FUNCTION_BLOCK FB_Estacion
VAR_INPUT
END_VAR
VAR_OUTPUT
	//Parametros de salida
	PaleCodigo: BYTE;
END_VAR
VAR
	//Entradas comunes
	PulsadorEmergencia AT %I*: BOOL;
    SelectorManual AT %I*: BOOL;
    PulsadorMarcha AT %I*: BOOL;
    PulsadorParada AT %I*: BOOL := TRUE; // Contacto normalmente cerrado
    EstacionConectada AT %I*: BOOL := TRUE;
    DetectorPresion AT %I*: BOOL := TRUE;
	
	PalePresencia AT %I*: BOOL;
    PaleCodigoBit0 AT %I*: BOOL;
    PaleCodigoBit1 AT %I*: BOOL;
    PaleCodigoBit2 AT %I*: BOOL;
	
	//Entradas específicas
	DescargadorDetras AT %I*: BOOL;
	DescargadorDelante AT %I*: BOOL;
	VerticalArriba AT %I*: BOOL;
	VerticalAbajo AT %I*: BOOL;
	VerificadorArriba AT %I*: BOOL;
	VerificadorAbajo AT %I*: BOOL;
	DesplazadorDetras AT %I*: BOOL;
	AlimentadorDetras AT %I*: BOOL;
	AlimentadorDelante AT %I*: BOOL;
	VacioDescargador AT %I*: BOOL;
	PresenciaBaseAlimentador AT %I*:BOOL;
	
	//Salidas comunes
	DesconectaEstacion AT %Q*: BOOL;
    LamparaAlarma AT %Q*: BOOL;
    LamparaMarcha AT %Q*: BOOL;
	LamparaFaltaMaterial AT %Q*: BOOL;
    AvisadorSonoro AT %Q*: BOOL;

    CintaMotorActiva AT %Q*: BOOL;
    CintaMotorInvierte AT %Q*: BOOL;
    CintaRetenedorBaja AT %Q*: BOOL;
    CintaSeparadorSube AT %Q*: BOOL;
	
	//Salidas específicas
	DescargadorAtras AT %Q*: BOOL;
	DescargadorAdelante AT %Q*: BOOL;
	DescargadorBaja AT %Q*: BOOL;
	RechazadorAdelante AT %Q*: BOOL;
	VerificadorBaja AT %Q*: BOOL;
	DesplazadorAdelante AT %Q*: BOOL;
	AlimentadorAdelante AT %Q*: BOOL;
	EyectorSucciona AT %Q*: BOOL;
END_VAR

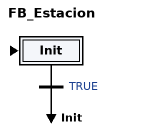
INITIAL_STEP Init:
END_STEP
TRANSITION FROM Init TO Init
    := TRUE;
END_TRANSITION

ACTION aPaleCodigo:
PaleCodigo.0 := PaleCodigoBit0;
PaleCodigo.1 := PaleCodigoBit1;
PaleCodigo.2 := PaleCodigoBit2;
END_ACTION

END_FUNCTION_BLOCK

(* stored: Version 1.1.0.1, ProductVersion 3.1.4024.12
   POU FB_Estacion: Id {ec7f9724-88c9-49d4-878c-113169f296e7}, SpecialFunc None
   Action aPaleCodigo: Id {1981cdec-f364-46d7-8928-81208a9a2e3d} *)
